TYPE structAlarm :
STRUCT
	xAlarmIN	:	BOOL;	//Alarm Trigger
	xAlarmOFF	:	BOOL;	//Alarm übersteuert (wird nicht ausgelöst)
	xAlarmSAVE	:	BOOL;	//Alarm gespeichert (muss quittiert werden)
	xAlarmQUIT	:	BOOL;	//Alarm quittieren
	xAlarmOUT	:	BOOL;	//Alarm aktiv
	tAlarmVERZ	:	TIME;	//Alarmverzögerung
	sAlarmText	:	STRING;	//Alarmtext
	bAlarmNr	:	BYTE;	//Zusatztext #
END_STRUCT
END_TYPE

(* stored: Version 1.1.0.1, ProductVersion 3.1.4024.6
   DUT structAlarm: Id {6b132e64-cfc8-4c5d-bbb8-486ab5c40044} *)
